// TIA Portal V16 export
// export: Created 2023-03-29T11:03:42.2880272Z, ExportSetting WithDefaults, DisplayName Totally Integrated Automation Portal, DisplayVersion V16 Update 6, DisplayName TIA Portal Version Control Interface, DisplayVersion V16 Update 2, DisplayName TIA Portal Openness, DisplayVersion V16 Update 6, DisplayName STEP 7 Professional, DisplayVersion V16 Update 6, DisplayName STEP 7 Safety, DisplayVersion V16, DisplayName WinCC Advanced, DisplayVersion V16 Update 6
DATA_BLOCK "dbtags_Sterowanie"   // DB1
{ S7_Optimized_Access := 'FALSE' }
VERSION : 0.1
// stored: AutoNumber false, DBAccessibleFromOPCUA true, IsOnlyStoredInLoadMemory false, IsWriteProtectedInAS false
   VAR RETAIN
      HMI : Struct
         PhysicalUnit : String[5] := '1/min';
         Output_PWM_USInt : USInt;
         "position reached" : Bool;   // bit potwierdzenia zasuwa Z10 na pozycji
         ManualMode_visible : Bool;
         Manual_ : Bool;   // rez
         ErrorAck_1_Int : Int;
         ErrorAck_Int : Int;
         Warning_Int : Int;
         ErrorAck_Int_edge : Bool;
         ErrorAck : Bool;
         Acknowledge_visible : Bool;
         resetScreen_1 : Bool;
         resetScreen_2 : Bool := false;
         resetScreen_3 : Bool := false;
         resetScreen_4 : Bool := false;
         resetScreen_5 : Bool := false;
         resetScreen_6 : Bool := false;
         resetScreen_7 : Bool := false;
         resetScreen_8 : Bool := false;
         resetScreen_9 : Bool := false;
         resetScreen_10 : Bool := false;
         resetScreen_11 : Bool := false;
         resetScreen_12 : Bool := false;
         resetScreen_13 : Bool := false;
      END_STRUCT;
      "Z10 Pozycja" : Struct
         encoder : Word;
         rpm : Word;
      END_STRUCT;
      SetupControl : Struct
         Static_ : Bool;
      END_STRUCT;
      "Analog pomiar" : Struct
         ciśnienie_B5 : Real;
         kolman_poziom_zbiornik_1 : Real;
         kolman_poziom_zbiornik_2 : Real := 16#0;
         kolman_poziom_zbiornik_3 : Real := 16#0;
         kolman_poziom_zbiornik_4 : Real := 16#0;
         AI_ciśnienie_B5 : Real;
         AI_poziom_zbiornik_1 : Real;
         AI_poziom_zbiornik_2 : Real := 0.0;
         AI_poziom_zbiornik_3 : Real := 0.0;
         AI_poziom_zbiornik_4 : Real := 0.0;
      END_STRUCT;
   END_VAR
BEGIN
END_DATA_BLOCK
